PROGRAM OP130_LH_Auto
VAR
	OP130_Torque_Monitor_Dly: TON;
	Temp1:BOOL;
	act_torque:LREAL;
END_VAR

CASE OP130_LH_AutoSeq OF
	10: IF (OP130_Prev_LH_COMP_OK= TRUE) AND OP130_StartEnable THEN   //Check LH Comp OK
		OP130_LH_AutoSeq:=20;
		END_IF
		IF (OP130_Prev_LH_COMP_NOK= TRUE) THEN 
			OP130_LH_AutoSeq:=180;
		END_IF
	
	20:IF  OP130_StartEnable THEN	// Check Mover Presence in Station
		   OP130_LH_AutoSeq:=30;
	   END_IF
	   
	30:IF (OP130_GVL.SR130_LH_Servo_Control.Axis_Enabled=TRUE OR OP130_Dry_Run) AND OP130_StartEnable THEN // Check Servo Axis Enabled
		   OP130_LH_AutoSeq:=40;
		END_IF
		
	40:IF  OP130_StartEnable THEN  // Check Rotary Cyl In Zero Deg
		   OP130_LH_AutoSeq:=50;
	   END_IF
	   
	50:IF OP130_StartEnable THEN 		//Move Work Position Value to Servo
		//  OP130_GVL.SR130_LH_Vert_Servo.fTargetPosition:=SR130_HMI_Servo_Work_Position;
		//  OP130_GVL.SR130_LH_Vert_Servo.fTargetVelocity:=SR130_HMI_Servo_Work_Velocity;
		SR130_LH_Servo_Control.Position:=SR130_HMI_Servo_Work_Position;
		SR130_LH_Servo_Control.Velocity:=SR130_HMI_Servo_Work_Velocity;
		OP130_LH_AutoSeq:=60;
		END_IF
		
	60:IF OP130_StartEnable THEN 	//Move Cmd to Servo
		//SR130_LH_Abs_Move_Start:=TRUE;
		SR130_LH_Servo_Control.ABSmove_Start:=TRUE;
		OP130_LH_AutoSeq:=70;
		END_IF
		
	70:IF OP130_StartEnable AND OP130_GVL.SR130_LH_Servo_Control.Axis_In_Pos THEN // Check Servo in Target Pos
		//SR130_LH_Abs_Move_Start:=FALSE;
		SR130_LH_Servo_Control.ABSmove_Start:=FALSE;
		OP130_LH_AutoSeq:=90;
		END_IF
	
	90:IF OP130_StartEnable THEN		//Move Lock Position Value to Servo
		//OP130_GVL.SR130_LH_Vert_Servo.fTargetPosition:=SR130_HMI_Servo_Lock_Position;
		//OP130_GVL.SR130_LH_Vert_Servo.fTargetVelocity:=SR130_HMI_Servo_Lock_Velocity;
	     SR130_LH_Servo_Control.Position:=SR130_HMI_Servo_Lock_Position;
		 SR130_LH_Servo_Control.Velocity:=SR130_HMI_Servo_Lock_Velocity;
		 OP130_LH_AutoSeq:=100;
		 END_IF
		 
	100:IF OP130_StartEnable THEN		// MOve Cmd to Servo
		//SR130_LH_Abs_Move_Start:=TRUE;
		   SR130_LH_Servo_Control.ABSmove_Start :=TRUE;
		   OP130_LH_AutoSeq:=110;
		END_IF
		
    110:IF OP130_StartEnable  THEN		//Check Servo In Target Pos
		IF SR130_LH_Servo_Control.Axis_In_Pos AND SR130_LH_Servo_Control.Actual_Torque < OP130_HMI_Pull_Torque_Limit THEN
			act_torque:=SR130_LH_Servo_Control.Actual_Torque;
			SR130_LH_Vert_Servo.bHalt:=TRUE;
			OP130_LH_Comp_OK:=TRUE;
			OP130_LH_Comp_NOK:= FALSE;
	//	SR130_LH_Abs_Move_Start:=FALSE;
		SR130_LH_Servo_Control.ABSmove_Start:=FALSE;
		END_IF
		IF SR130_LH_Servo_Control.Axis_In_Pos AND SR130_LH_Servo_Control.Actual_Torque > OP130_HMI_Pull_Torque_Limit THEN
			OP130_LH_Comp_NOK:=TRUE;
			OP130_LH_Comp_OK:= FALSE;
			//SR130_LH_Abs_Move_Start:=FALSE;
			SR130_LH_Servo_Control.ABSmove_Start:=FALSE;
		END_IF
	    IF SR130_LH_Servo_Control.Axis_Halted OR SR130_LH_Servo_Control.Axis_In_Pos AND (OP130_LH_Comp_OK OR OP130_LH_Comp_NOK) THEN
	    //SR130_LH_Abs_Move_Start:=FALSE;
		SR130_LH_Servo_Control.ABSmove_Start:=FALSE;
        OP130_LH_AutoSeq:=180;
	    END_IF
        END_IF
	
		

	
	180:IF (OP130_StartEnable) THEN   // Move Work Pos Values to Servo
		//OP130_GVL.SR130_LH_Vert_Servo.fTargetPosition:=SR130_HMI_Servo_CylWork_Position;
       // OP130_GVL.SR130_LH_Vert_Servo.fTargetVelocity:=SR130_HMI_Servo_CylWork_Velocity;
		SR130_LH_Servo_Control.position:=SR130_HMI_Servo_CylWork_Position;
		SR130_LH_Servo_Control.velocity:=SR130_HMI_Servo_CylWork_Velocity;
		SR130_LH_Vert_Servo.bHalt:=FALSE;
        MOVER_CMP_STATUS[OP130_STN_MOVER][1]:=130;
        OP130_LH_AutoSeq:=190;
	   END_IF
	   
	 190: IF(OP130_StartEnable) THEN		//move Cmd to Servo
		// SR130_LH_Abs_Move_Start:= TRUE;
		 SR130_LH_Servo_Control.ABSmove_Start := TRUE;
		 OP130_LH_AutoSeq:=200;
	 END_IF
	 
	200:IF (OP130_StartEnable) AND OP130_GVL.SR130_LH_Servo_Control.Axis_In_Pos THEN		//Check Servo In Target Pos
	       //SR130_LH_Abs_Move_Start:= FALSE;	
		   SR130_LH_Servo_Control.ABSmove_Start := FALSE;
           OP130_LH_AutoSeq:=210;
	    END_IF
		
	210:IF  (OP130_StartEnable) THEN		//Move Rotary Cyl to Zero Deg
		    OP130_GVL.CR130_LH_Rot_Cyl.AutoCmd2:=TRUE;
		    OP130_GVL.CR130_LH_Rot_Cyl.AutoCmd1:=FALSE;
		    IF (OP130_GVL.CR130_LH_Rot_Cyl.Position2=TRUE) THEN
			   OP130_LH_AutoSeq:=220;
			   END_IF
	    END_IF
		
	220: IF  (OP130_StartEnable) THEN		//move Home Pos to Servo
		    // OP130_GVL.SR130_LH_Vert_Servo.fTargetPosition:=SR130_HMI_Servo_Rotation_Position;
		    // OP130_GVL.SR130_LH_Vert_Servo.fTargetVelocity:=SR130_HMI_Servo_Rotation_Velocity;
			 SR130_LH_Servo_Control.Position :=SR130_HMI_Servo_Rotation_Position;
			 SR130_LH_Servo_Control.Velocity :=SR130_HMI_Servo_Rotation_Velocity;
		     OP130_LH_AutoSeq:=230;
	      END_IF
	
	230: IF (OP130_StartEnable) THEN 		//Move Cmd TO Servo
		   // SR130_LH_Abs_Move_Start:= TRUE ;
			SR130_LH_Servo_Control.ABSmove_Start:= TRUE;
		    OP130_LH_AutoSeq:=240;
	     END_IF
	
	240: IF (OP130_StartEnable) AND OP130_GVL.SR130_LH_Servo_Control.Axis_In_Pos THEN 	//Check Servo In Target Pos
		    //SR130_LH_Abs_Move_Start:= FALSE ;
			SR130_LH_Servo_Control.ABSmove_Start:= FALSE;
			OP130_LH_AutoSeq:=250;
	     END_IF
	
	250:IF  (OP130_StartEnable) THEN		//Move Rotary Cyl to Zero Deg
		    OP130_GVL.CR130_LH_Rot_Cyl.AutoCmd1:=TRUE;
		    OP130_GVL.CR130_LH_Rot_Cyl.AutoCmd2:=FALSE;
		   IF (OP130_GVL.CR130_LH_Rot_Cyl.Position1=TRUE) THEN
			  OP130_LH_AutoSeq:=260;
		   END_IF
	    END_IF
		
	260: IF  (OP130_StartEnable) THEN		//move Home Pos to Servo
		     //OP130_GVL.SR130_LH_Vert_Servo.fTargetPosition:=SR130_Servo_Home_Position;
		    // OP130_GVL.SR130_LH_Vert_Servo.fTargetVelocity:=SR130_Servo_Home_Velocity;
			 SR130_LH_Servo_Control.Position := SR130_Servo_Home_Position;
			 SR130_LH_Servo_Control.Velocity := SR130_Servo_Home_Velocity;
		     OP130_LH_AutoSeq:=270;
	     END_IF
		 
	270: IF (OP130_StartEnable) THEN 		//Move Cmd TO Servo
		   // SR130_LH_Abs_Move_Start:= TRUE ;
			SR130_LH_Servo_Control.ABSmove_Start := TRUE;
		    OP130_LH_AutoSeq:=280;
	     END_IF
	
	280: IF (OP130_StartEnable) AND OP130_GVL.SR130_LH_Servo_Control.Axis_In_Pos THEN 	//Check Servo In Target Pos
		   // SR130_LH_Abs_Move_Start:= FALSE ;
			SR130_LH_Servo_Control.ABSmove_Start := FALSE;
			OP130_LH_AutoSeq:=290;
	     END_IF
		 
	 290:IF (OP130_StartEnable) THEN		//LH Operation completed
		    OP130_LH_Operation_Completed:= TRUE;
		    OP130_LH_AutoSeq:=300;
	     END_IF

	   
END_CASE
//Torque Monitor Delay
OP130_Torque_Monitor_Dly(IN:=OP130_LH_AutoSeq=170 , PT:=T#200MS , Q=> , ET=> );

END_PROGRAM

(* stored: Version 1.1.0.1, ProductVersion 3.1.4024.11
   POU OP130_LH_Auto: Id {07c888b9-abf3-414e-9fbe-2377212607a7}, SpecialFunc None *)
